// TIA Portal V17 export
// export: Created 2025-03-07T09:18:41.3441384Z, ExportSetting WithDefaults, DisplayName Totally Integrated Automation Portal, DisplayVersion V17 Update 8, DisplayName TIA Portal Openness, DisplayVersion V17 Update 8, DisplayName TIA Portal Version Control Interface, DisplayVersion V17, DisplayName SINAMICS Startdrive Advanced, DisplayVersion V17 SP2, DisplayName SINAMICS Startdrive G110M, G120, G120C, G120D, G120P, G115D, DisplayVersion V17 SP2, DisplayName SINAMICS Startdrive G130, G150, S120, S150, SINAMICS MV, S210, DisplayVersion V17 SP2, DisplayName STEP 7 Professional, DisplayVersion V17 Update 8, DisplayName SINUMERIK ONE STEP 7 Toolbox, DisplayVersion V17 Update 12, DisplayName SINUMERIK 840D sl STEP 7 Toolbox, DisplayVersion V17 Update 12, DisplayName STEP 7 Safety, DisplayVersion V17 Update 6, DisplayName WinCC Advanced, DisplayVersion V17 Update 8
DATA_BLOCK "DB1041_C11_BRAKE_TEST"   // DB1041
{ DB_Accessible_From_OPC_UA := 'FALSE' }
AUTHOR : ETXETAR
VERSION : 1.0
// stored: AutoNumber false, DBAccessibleFromOPCUA false, DBAccessibleFromWebserver true, InstanceOfName FB1031_BRAKE_TEST, InstanceOfType FB
"FB1031_BRAKE_TEST"
   // VAR_INPUT
   //    START_REQ : Bool;
   //    BRAKE_SELECT : Bool;
   //    DIRECTION_OF_ROT : Bool;
   //    TORQUE_SELECT : Bool;
   //    "BRAKE_CLOSED(ONLY EXTERNAL)" : Bool;
   // END_VAR
   // VAR_OUTPUT
   //    BRAKE_TEST_ACTIVE : Bool;
   //    BRAKE_TEST_DONE : Bool;
   //    BRAKE_TEST_ERROR : Bool;
   //    SELECTED_BRAKE : Bool;
   //    "BRAKE_REQ(ONLY_EXTERNAL)" : Bool;
   //    SIGN_OF_LOAD : Bool;
   // END_VAR
   // VAR_IN_OUT
   //    AXIS_DB : "LBP_typeAxisX";
   // END_VAR
   // VAR RETAIN
   //    Timer_Brake_test_DONE { ExternalAccessible := 'False'; ExternalVisible := 'False'; ExternalWritable := 'False'; S7_SetPoint := 'True'} : TON_TIME;
   //    Timer_Brake_test_ERROR { ExternalAccessible := 'False'; ExternalVisible := 'False'; ExternalWritable := 'False'; S7_SetPoint := 'True'} : TON_TIME;
   // END_VAR
BEGIN
END_DATA_BLOCK
